KUKA KRL program: nplacestr5LS1.src, nplacestr5LS1.dat

--- nplacestr5LS1.src ---
&ACCESS RVP
&REL 1
&PARAM TEMPLATE = C:\KRC\Roboter\Template\ExpertVorgabe
&PARAM EDITMASK = *
DEF nplacestr5LS1( )
;FOLD INI
  ;FOLD BASISTECH INI
    GLOBAL INTERRUPT DECL 3 WHEN $STOPMESS==TRUE DO IR_STOPM ( )
    INTERRUPT ON 3
    BAS (#INITMOV,0 )
  ;ENDFOLD (BASISTECH INI)
  ;FOLD USER INI
    ;Make your modifications here

  ;ENDFOLD (USER INI)
;ENDFOLD (INI)




SWITCH NumCuring

;*******************************************************
CASE 90501
;*******************************************************
;*** Utilizar para hacer touchup en ptp a continuacion ***;
; 1  Ejecutar Axis_Rob_Move
; 2  Hacer TouchUp en ptp
; 3  Eliminar Axis_Rob_Move y comentarios

Axis_Rob_Move(1.69,-82.8,66.93,14.32,12.14,193,70,50)

;FOLD PTP pWB90501LS1 Vel=100 % PDAT_MESA Tool[10]:AMF1_G1000 Base[14]:BWB2S1;%{PE}%R 5.5.32,%MKUKATPBASIS,%CMOVE,%VPTP,%P 1:PTP, 2:pWB90501LS1, 3:, 5:100, 7:PDAT_MESA
$BWDSTART=FALSE
PDAT_ACT=PPDAT_MESA
FDAT_ACT=FpWB90501LS1
BAS(#PTP_PARAMS,100)
PTP XpWB90501LS1
;ENDFOLD
;*********************************************************;

;***Axis_Rob_Move de ayuda para aproximarse a dejada ***;
; Borrar tras touchup en LIN de dejada
Axis_Rob_Move(-90.22,-57.13,49.23,-5.44,97.37,193.9,20,50)
;*******************************************************;

PTP_OFFS(XP90501LS1, FP90501LS1, 0, -450, 30, 0, 0, 0, #TOOL, 20, 50, 0.0)

Cicle_Grp_M1000 (Inic_Pla_Right)

;***borrar***;
cyltopos(prg_200)
halt
;************;

LIN_OFFS(XP90501LS1, FP90501LS1, 0, 0, 30, 0, 0, 0, #TOOL, 0.1, 50, 0.0)
LIN_OFFS(XP90501LS1, FP90501LS1, 0, 0, 15, 0, 0, 0, #TOOL, 0.1, 50, 0.0)

Cntr_Grp_M1000 (C05C06,RH)

;FOLD LIN P90501LS1 Vel=0.1 m/s LV020Z0 Tool[10]:AMF1_G1000 Base[14]:BWB2S1;%{PE}%R 5.5.32,%MKUKATPBASIS,%CMOVE,%VLIN,%P 1:LIN, 2:P90501LS1, 3:, 5:0.1, 7:V020Z0
$BWDSTART=FALSE
LDAT_ACT=LV020Z0
FDAT_ACT=FP90501LS1
BAS(#CP_PARAMS,0.1)
LIN XP90501LS1
;ENDFOLD

Cntr_Grp_M1000 (AMF09,RLS)
Cyltopos (PRG_51)
Cntr_Grp_M1000 (C07C08,RH)
Cyltopos (PRG_61)
Cntr_Grp_M1000 (AMF10,RLS)
Cntr_Grp_M1000 (C05C06,FREE)
Cntr_Grp_M1000 (C07C08,FREE)
Cyltopos(PRG_88)
LIN_REL{Z -20}#TOOL
Cyltopos (PRG_105)
LIN_REL{Z -30}#TOOL
Cyltopos (PRG_200)

;*** MOVIMIENTOS DE OFFSETS ***;

LIN_OFFS(XP90501LS1, FP90501LS1, 0, 0, -50, 0, 0, 0, #TOOL, 0.3, 50, 0.0)
LIN_OFFS(XP90501LS1, FP90501LS1, 0, -450, -50, 0, 0, 0, #TOOL, 0.3, 50, 0.0)


;******* MEDICION LASER *******;

LIN_OFFS(XPLAS90501LS1_1, FPLAS90501LS1_1, 0, -200, 0, 0, 0, 0, #TOOL, 0.3, 50, 0.0)

cyltopos (prg_61)

;FOLD LIN PLAS90501LS1_1 Vel=0.3 m/s LV020Z0 Tool[10]:AMF1_G1000 Base[14]:BWB2S1;%{PE}%R 5.5.32,%MKUKATPBASIS,%CMOVE,%VLIN,%P 1:LIN, 2:PLAS90501LS1_1, 3:, 5:0.3, 7:V020Z0
$BWDSTART=FALSE
LDAT_ACT=LV020Z0
FDAT_ACT=FPLAS90501LS1_1
BAS(#CP_PARAMS,0.3)
LIN XPLAS90501LS1_1
;ENDFOLD

;Movimimiento de busqueda con laser
;Search( , )

;FOLD LIN PLAS90501LS1_2 Vel=0.3 m/s LV020Z0 Tool[10]:AMF1_G1000 Base[14]:BWB2S1;%{PE}%R 5.5.32,%MKUKATPBASIS,%CMOVE,%VLIN,%P 1:LIN, 2:PLAS90501LS1_2, 3:, 5:0.3, 7:V020Z0
$BWDSTART=FALSE
LDAT_ACT=LV020Z0
FDAT_ACT=FPLAS90501LS1_2
BAS(#CP_PARAMS,0.3)
LIN XPLAS90501LS1_2
;ENDFOLD


;Movimimiento de busqueda con laser
;Search( , )

LIN_OFFS(XPLAS90501LS1_1, FPLAS90501LS1_1, 0, -200, 0, 0, 0, 0, #TOOL, 0.3, 50, 0.0)

;******************************;

;FOLD PTP pWB90501LS1 Vel=100 % PDAT_MESA Tool[10]:AMF1_G1000 Base[14]:BWB2S1;%{PE}%R 5.5.32,%MKUKATPBASIS,%CMOVE,%VPTP,%P 1:PTP, 2:pWB90501LS1, 3:, 5:100, 7:PDAT_MESA
$BWDSTART=FALSE
PDAT_ACT=PPDAT_MESA
FDAT_ACT=FpWB90501LS1
BAS(#PTP_PARAMS,100)
PTP XpWB90501LS1
;ENDFOLD

;*******************************************************
CASE 90503
;*******************************************************
;*** Utilizar para hacer touchup en ptp a continuacion ***;
; 1  Ejecutar Axis_Rob_Move
; 2  Hacer TouchUp en ptp
; 3  Eliminar Axis_Rob_Move y comentarios

Axis_Rob_Move(1.69,-82.8,66.93,14.32,12.14,193,70,50)

;FOLD PTP pWB90503LS1 Vel=100 % PDAT_MESA Tool[10]:AMF1_G1000 Base[14]:BWB2S1;%{PE}%R 5.5.32,%MKUKATPBASIS,%CMOVE,%VPTP,%P 1:PTP, 2:pWB90503LS1, 3:, 5:100, 7:PDAT_MESA
$BWDSTART=FALSE
PDAT_ACT=PPDAT_MESA
FDAT_ACT=FpWB90503LS1
BAS(#PTP_PARAMS,100)
PTP XpWB90503LS1
;ENDFOLD
;*********************************************************;

;***Axis_Rob_Move de ayuda para aproximarse a dejada ***;
; Borrar tras touchup en LIN de dejada
Axis_Rob_Move(-90.22,-57.13,49.23,-5.44,97.37,193.9,20,50)
;*******************************************************;

PTP_OFFS(XP90503LS1, FP90503LS1, 0, -450, 30, 0, 0, 0, #TOOL, 20, 50, 0.0)

Cicle_Grp_M1000 (Inic_Pla_Right)

;***borrar***;
cyltopos(prg_200)
halt
;************;

LIN_OFFS(XP90503LS1, FP90503LS1, 0, 0, 30, 0, 0, 0, #TOOL, 0.1, 50, 0.0)
LIN_OFFS(XP90503LS1, FP90503LS1, 0, 0, 15, 0, 0, 0, #TOOL, 0.1, 50, 0.0)

Cntr_Grp_M1000 (C05C06,RH)

;FOLD LIN P90503LS1 Vel=0.1 m/s LV020Z0 Tool[10]:AMF1_G1000 Base[14]:BWB2S1;%{PE}%R 5.5.32,%MKUKATPBASIS,%CMOVE,%VLIN,%P 1:LIN, 2:P90503LS1, 3:, 5:0.1, 7:V020Z0
$BWDSTART=FALSE
LDAT_ACT=LV020Z0
FDAT_ACT=FP90503LS1
BAS(#CP_PARAMS,0.1)
LIN XP90503LS1
;ENDFOLD

Cntr_Grp_M1000 (AMF09,RLS)
Cyltopos (PRG_51)
Cntr_Grp_M1000 (C07C08,RH)
Cyltopos (PRG_61)
Cntr_Grp_M1000 (AMF10,RLS)
Cntr_Grp_M1000 (C05C06,FREE)
Cntr_Grp_M1000 (C07C08,FREE)
Cyltopos(PRG_88)
LIN_REL{Z -20}#TOOL
Cyltopos (PRG_105)
LIN_REL{Z -30}#TOOL
Cyltopos (PRG_200)

;*** MOVIMIENTOS DE OFFSETS ***;

LIN_OFFS(XP90503LS1, FP90503LS1, 0, 0, -50, 0, 0, 0, #TOOL, 0.3, 50, 0.0)
LIN_OFFS(XP90503LS1, FP90503LS1, 0, -450, -50, 0, 0, 0, #TOOL, 0.3, 50, 0.0)


;******* MEDICION LASER *******;

LIN_OFFS(XPLAS90503LS1_1, FPLAS90503LS1_1, 0, -200, 0, 0, 0, 0, #TOOL, 0.3, 50, 0.0)

cyltopos (prg_61)

;FOLD LIN PLAS90503LS1_1 Vel=0.3 m/s LV020Z0 Tool[10]:AMF1_G1000 Base[14]:BWB2S1;%{PE}%R 5.5.32,%MKUKATPBASIS,%CMOVE,%VLIN,%P 1:LIN, 2:PLAS90503LS1_1, 3:, 5:0.3, 7:V020Z0
$BWDSTART=FALSE
LDAT_ACT=LV020Z0
FDAT_ACT=FPLAS90503LS1_1
BAS(#CP_PARAMS,0.3)
LIN XPLAS90503LS1_1
;ENDFOLD

;Movimimiento de busqueda con laser
;Search( , )

;FOLD LIN PLAS90503LS1_2 Vel=0.3 m/s LV020Z0 Tool[10]:AMF1_G1000 Base[14]:BWB2S1;%{PE}%R 5.5.32,%MKUKATPBASIS,%CMOVE,%VLIN,%P 1:LIN, 2:PLAS90503LS1_2, 3:, 5:0.3, 7:V020Z0
$BWDSTART=FALSE
LDAT_ACT=LV020Z0
FDAT_ACT=FPLAS90503LS1_2
BAS(#CP_PARAMS,0.3)
LIN XPLAS90503LS1_2
;ENDFOLD


;Movimimiento de busqueda con laser
;Search( , )

LIN_OFFS(XPLAS90503LS1_1, FPLAS90503LS1_1, 0, -200, 0, 0, 0, 0, #TOOL, 0.3, 50, 0.0)

;******************************;

;FOLD PTP pWB90503LS1 Vel=100 % PDAT_MESA Tool[10]:AMF1_G1000 Base[14]:BWB2S1;%{PE}%R 5.5.32,%MKUKATPBASIS,%CMOVE,%VPTP,%P 1:PTP, 2:pWB90503LS1, 3:, 5:100, 7:PDAT_MESA
$BWDSTART=FALSE
PDAT_ACT=PPDAT_MESA
FDAT_ACT=FpWB90503LS1
BAS(#PTP_PARAMS,100)
PTP XpWB90503LS1
;ENDFOLD

;*******************************************************
CASE 90505
;*******************************************************
;*** Utilizar para hacer touchup en ptp a continuacion ***;
; 1  Ejecutar Axis_Rob_Move
; 2  Hacer TouchUp en ptp
; 3  Eliminar Axis_Rob_Move y comentarios

Axis_Rob_Move(1.69,-82.8,66.93,14.32,12.14,193,70,50)

;FOLD PTP pWB90505LS1 Vel=100 % PDAT_MESA Tool[10]:AMF1_G1000 Base[14]:BWB2S1;%{PE}%R 5.5.32,%MKUKATPBASIS,%CMOVE,%VPTP,%P 1:PTP, 2:pWB90505LS1, 3:, 5:100, 7:PDAT_MESA
$BWDSTART=FALSE
PDAT_ACT=PPDAT_MESA
FDAT_ACT=FpWB90505LS1
BAS(#PTP_PARAMS,100)
PTP XpWB90505LS1
;ENDFOLD
;*********************************************************;

;***Axis_Rob_Move de ayuda para aproximarse a dejada ***;
; Borrar tras touchup en LIN de dejada
Axis_Rob_Move(-90.22,-57.13,49.23,-5.44,97.37,193.9,20,50)
;*******************************************************;

PTP_OFFS(XP90505LS1, FP90505LS1, 0, -450, 30, 0, 0, 0, #TOOL, 20, 50, 0.0)

Cicle_Grp_M1000 (Inic_Pla_Right)

;***borrar***;
cyltopos(prg_200)
halt
;************;

LIN_OFFS(XP90505LS1, FP90505LS1, 0, 0, 30, 0, 0, 0, #TOOL, 0.1, 50, 0.0)
LIN_OFFS(XP90505LS1, FP90505LS1, 0, 0, 15, 0, 0, 0, #TOOL, 0.1, 50, 0.0)

Cntr_Grp_M1000 (C05C06,RH)

;FOLD LIN P90505LS1 Vel=0.1 m/s LV020Z0 Tool[10]:AMF1_G1000 Base[14]:BWB2S1;%{PE}%R 5.5.32,%MKUKATPBASIS,%CMOVE,%VLIN,%P 1:LIN, 2:P90505LS1, 3:, 5:0.1, 7:V020Z0
$BWDSTART=FALSE
LDAT_ACT=LV020Z0
FDAT_ACT=FP90505LS1
BAS(#CP_PARAMS,0.1)
LIN XP90505LS1
;ENDFOLD

Cntr_Grp_M1000 (AMF09,RLS)
Cyltopos (PRG_51)
Cntr_Grp_M1000 (C07C08,RH)
Cyltopos (PRG_61)
Cntr_Grp_M1000 (AMF10,RLS)
Cntr_Grp_M1000 (C05C06,FREE)
Cntr_Grp_M1000 (C07C08,FREE)
Cyltopos(PRG_88)
LIN_REL{Z -20}#TOOL
Cyltopos (PRG_105)
LIN_REL{Z -30}#TOOL
Cyltopos (PRG_200)

;*** MOVIMIENTOS DE OFFSETS ***;

LIN_OFFS(XP90505LS1, FP90505LS1, 0, 0, -50, 0, 0, 0, #TOOL, 0.3, 50, 0.0)
LIN_OFFS(XP90505LS1, FP90505LS1, 0, -450, -50, 0, 0, 0, #TOOL, 0.3, 50, 0.0)


;******* MEDICION LASER *******;

LIN_OFFS(XPLAS90505LS1_1, FPLAS90505LS1_1, 0, -200, 0, 0, 0, 0, #TOOL, 0.3, 50, 0.0)

cyltopos (prg_61)

;FOLD LIN PLAS90505LS1_1 Vel=0.3 m/s LV020Z0 Tool[10]:AMF1_G1000 Base[14]:BWB2S1;%{PE}%R 5.5.32,%MKUKATPBASIS,%CMOVE,%VLIN,%P 1:LIN, 2:PLAS90505LS1_1, 3:, 5:0.3, 7:V020Z0
$BWDSTART=FALSE
LDAT_ACT=LV020Z0
FDAT_ACT=FPLAS90505LS1_1
BAS(#CP_PARAMS,0.3)
LIN XPLAS90505LS1_1
;ENDFOLD

;Movimimiento de busqueda con laser
;Search( , )

;FOLD LIN PLAS90505LS1_2 Vel=0.3 m/s LV020Z0 Tool[10]:AMF1_G1000 Base[14]:BWB2S1;%{PE}%R 5.5.32,%MKUKATPBASIS,%CMOVE,%VLIN,%P 1:LIN, 2:PLAS90505LS1_2, 3:, 5:0.3, 7:V020Z0
$BWDSTART=FALSE
LDAT_ACT=LV020Z0
FDAT_ACT=FPLAS90505LS1_2
BAS(#CP_PARAMS,0.3)
LIN XPLAS90505LS1_2
;ENDFOLD


;Movimimiento de busqueda con laser
;Search( , )

LIN_OFFS(XPLAS90505LS1_1, FPLAS90505LS1_1, 0, -200, 0, 0, 0, 0, #TOOL, 0.3, 50, 0.0)

;******************************;

;FOLD PTP pWB90505LS1 Vel=100 % PDAT_MESA Tool[10]:AMF1_G1000 Base[14]:BWB2S1;%{PE}%R 5.5.32,%MKUKATPBASIS,%CMOVE,%VPTP,%P 1:PTP, 2:pWB90505LS1, 3:, 5:100, 7:PDAT_MESA
$BWDSTART=FALSE
PDAT_ACT=PPDAT_MESA
FDAT_ACT=FpWB90505LS1
BAS(#PTP_PARAMS,100)
PTP XpWB90505LS1
;ENDFOLD

;*******************************************************
CASE 90507
;*******************************************************
;*** Utilizar para hacer touchup en ptp a continuacion ***;
; 1  Ejecutar Axis_Rob_Move
; 2  Hacer TouchUp en ptp
; 3  Eliminar Axis_Rob_Move y comentarios

Axis_Rob_Move(1.69,-82.8,66.93,14.32,12.14,193,70,50)

;FOLD PTP pWB90507LS1 Vel=100 % PDAT_MESA Tool[10]:AMF1_G1000 Base[14]:BWB2S1;%{PE}%R 5.5.32,%MKUKATPBASIS,%CMOVE,%VPTP,%P 1:PTP, 2:pWB90507LS1, 3:, 5:100, 7:PDAT_MESA
$BWDSTART=FALSE
PDAT_ACT=PPDAT_MESA
FDAT_ACT=FpWB90507LS1
BAS(#PTP_PARAMS,100)
PTP XpWB90507LS1
;ENDFOLD
;*********************************************************;

;***Axis_Rob_Move de ayuda para aproximarse a dejada ***;
; Borrar tras touchup en LIN de dejada
Axis_Rob_Move(-90.22,-57.13,49.23,-5.44,97.37,193.9,20,50)
;*******************************************************;

PTP_OFFS(XP90507LS1, FP90507LS1, 0, -450, 30, 0, 0, 0, #TOOL, 20, 50, 0.0)

Cicle_Grp_M1000 (Inic_Pla_Right)

;***borrar***;
cyltopos(prg_200)
halt
;************;

LIN_OFFS(XP90507LS1, FP90507LS1, 0, 0, 30, 0, 0, 0, #TOOL, 0.1, 50, 0.0)
LIN_OFFS(XP90507LS1, FP90507LS1, 0, 0, 15, 0, 0, 0, #TOOL, 0.1, 50, 0.0)

Cntr_Grp_M1000 (C05C06,RH)

;FOLD LIN P90507LS1 Vel=0.1 m/s LV020Z0 Tool[10]:AMF1_G1000 Base[14]:BWB2S1;%{PE}%R 5.5.32,%MKUKATPBASIS,%CMOVE,%VLIN,%P 1:LIN, 2:P90507LS1, 3:, 5:0.1, 7:V020Z0
$BWDSTART=FALSE
LDAT_ACT=LV020Z0
FDAT_ACT=FP90507LS1
BAS(#CP_PARAMS,0.1)
LIN XP90507LS1
;ENDFOLD

Cntr_Grp_M1000 (AMF09,RLS)
Cyltopos (PRG_51)
Cntr_Grp_M1000 (C07C08,RH)
Cyltopos (PRG_61)
Cntr_Grp_M1000 (AMF10,RLS)
Cntr_Grp_M1000 (C05C06,FREE)
Cntr_Grp_M1000 (C07C08,FREE)
Cyltopos(PRG_88)
LIN_REL{Z -20}#TOOL
Cyltopos (PRG_105)
LIN_REL{Z -30}#TOOL
Cyltopos (PRG_200)

;*** MOVIMIENTOS DE OFFSETS ***;

LIN_OFFS(XP90507LS1, FP90507LS1, 0, 0, -50, 0, 0, 0, #TOOL, 0.3, 50, 0.0)
LIN_OFFS(XP90507LS1, FP90507LS1, 0, -450, -50, 0, 0, 0, #TOOL, 0.3, 50, 0.0)


;******* MEDICION LASER *******;

LIN_OFFS(XPLAS90507LS1_1, FPLAS90507LS1_1, 0, -200, 0, 0, 0, 0, #TOOL, 0.3, 50, 0.0)

cyltopos (prg_61)

;FOLD LIN PLAS90507LS1_1 Vel=0.3 m/s LV020Z0 Tool[10]:AMF1_G1000 Base[14]:BWB2S1;%{PE}%R 5.5.32,%MKUKATPBASIS,%CMOVE,%VLIN,%P 1:LIN, 2:PLAS90507LS1_1, 3:, 5:0.3, 7:V020Z0
$BWDSTART=FALSE
LDAT_ACT=LV020Z0
FDAT_ACT=FPLAS90507LS1_1
BAS(#CP_PARAMS,0.3)
LIN XPLAS90507LS1_1
;ENDFOLD

;Movimimiento de busqueda con laser
;Search( , )

;FOLD LIN PLAS90507LS1_2 Vel=0.3 m/s LV020Z0 Tool[10]:AMF1_G1000 Base[14]:BWB2S1;%{PE}%R 5.5.32,%MKUKATPBASIS,%CMOVE,%VLIN,%P 1:LIN, 2:PLAS90507LS1_2, 3:, 5:0.3, 7:V020Z0
$BWDSTART=FALSE
LDAT_ACT=LV020Z0
FDAT_ACT=FPLAS90507LS1_2
BAS(#CP_PARAMS,0.3)
LIN XPLAS90507LS1_2
;ENDFOLD


;Movimimiento de busqueda con laser
;Search( , )

LIN_OFFS(XPLAS90507LS1_1, FPLAS90507LS1_1, 0, -200, 0, 0, 0, 0, #TOOL, 0.3, 50, 0.0)

;******************************;

;FOLD PTP pWB90507LS1 Vel=100 % PDAT_MESA Tool[10]:AMF1_G1000 Base[14]:BWB2S1;%{PE}%R 5.5.32,%MKUKATPBASIS,%CMOVE,%VPTP,%P 1:PTP, 2:pWB90507LS1, 3:, 5:100, 7:PDAT_MESA
$BWDSTART=FALSE
PDAT_ACT=PPDAT_MESA
FDAT_ACT=FpWB90507LS1
BAS(#PTP_PARAMS,100)
PTP XpWB90507LS1
;ENDFOLD

;*******************************************************
CASE 90509
;*******************************************************
;*** Utilizar para hacer touchup en ptp a continuacion ***;
; 1  Ejecutar Axis_Rob_Move
; 2  Hacer TouchUp en ptp
; 3  Eliminar Axis_Rob_Move y comentarios

Axis_Rob_Move(1.69,-82.8,66.93,14.32,12.14,193,70,50)

;FOLD PTP pWB90509LS1 Vel=100 % PDAT_MESA Tool[10]:AMF1_G1000 Base[14]:BWB2S1;%{PE}%R 5.5.32,%MKUKATPBASIS,%CMOVE,%VPTP,%P 1:PTP, 2:pWB90509LS1, 3:, 5:100, 7:PDAT_MESA
$BWDSTART=FALSE
PDAT_ACT=PPDAT_MESA
FDAT_ACT=FpWB90509LS1
BAS(#PTP_PARAMS,100)
PTP XpWB90509LS1
;ENDFOLD
;*********************************************************;

;***Axis_Rob_Move de ayuda para aproximarse a dejada ***;
; Borrar tras touchup en LIN de dejada
Axis_Rob_Move(-90.22,-57.13,49.23,-5.44,97.37,193.9,20,50)
;*******************************************************;

PTP_OFFS(XP90509LS1, FP90509LS1, 0, -450, 30, 0, 0, 0, #TOOL, 20, 50, 0.0)

Cicle_Grp_M1000 (Inic_Pla_Right)

;***borrar***;
cyltopos(prg_200)
halt
;************;

LIN_OFFS(XP90509LS1, FP90509LS1, 0, 0, 30, 0, 0, 0, #TOOL, 0.1, 50, 0.0)
LIN_OFFS(XP90509LS1, FP90509LS1, 0, 0, 15, 0, 0, 0, #TOOL, 0.1, 50, 0.0)

Cntr_Grp_M1000 (C05C06,RH)

;FOLD LIN P90509LS1 Vel=0.1 m/s LV020Z0 Tool[10]:AMF1_G1000 Base[14]:BWB2S1;%{PE}%R 5.5.32,%MKUKATPBASIS,%CMOVE,%VLIN,%P 1:LIN, 2:P90509LS1, 3:, 5:0.1, 7:V020Z0
$BWDSTART=FALSE
LDAT_ACT=LV020Z0
FDAT_ACT=FP90509LS1
BAS(#CP_PARAMS,0.1)
LIN XP90509LS1
;ENDFOLD

Cntr_Grp_M1000 (AMF09,RLS)
Cyltopos (PRG_51)
Cntr_Grp_M1000 (C07C08,RH)
Cyltopos (PRG_61)
Cntr_Grp_M1000 (AMF10,RLS)
Cntr_Grp_M1000 (C05C06,FREE)
Cntr_Grp_M1000 (C07C08,FREE)
Cyltopos(PRG_88)
LIN_REL{Z -20}#TOOL
Cyltopos (PRG_105)
LIN_REL{Z -30}#TOOL
Cyltopos (PRG_200)

;*** MOVIMIENTOS DE OFFSETS ***;

LIN_OFFS(XP90509LS1, FP90509LS1, 0, 0, -50, 0, 0, 0, #TOOL, 0.3, 50, 0.0)
LIN_OFFS(XP90509LS1, FP90509LS1, 0, -450, -50, 0, 0, 0, #TOOL, 0.3, 50, 0.0)


;******* MEDICION LASER *******;

LIN_OFFS(XPLAS90509LS1_1, FPLAS90509LS1_1, 0, -200, 0, 0, 0, 0, #TOOL, 0.3, 50, 0.0)

cyltopos (prg_61)

;FOLD LIN PLAS90509LS1_1 Vel=0.3 m/s LV020Z0 Tool[10]:AMF1_G1000 Base[14]:BWB2S1;%{PE}%R 5.5.32,%MKUKATPBASIS,%CMOVE,%VLIN,%P 1:LIN, 2:PLAS90509LS1_1, 3:, 5:0.3, 7:V020Z0
$BWDSTART=FALSE
LDAT_ACT=LV020Z0
FDAT_ACT=FPLAS90509LS1_1
BAS(#CP_PARAMS,0.3)
LIN XPLAS90509LS1_1
;ENDFOLD

;Movimimiento de busqueda con laser
;Search( , )

;FOLD LIN PLAS90509LS1_2 Vel=0.3 m/s LV020Z0 Tool[10]:AMF1_G1000 Base[14]:BWB2S1;%{PE}%R 5.5.32,%MKUKATPBASIS,%CMOVE,%VLIN,%P 1:LIN, 2:PLAS90509LS1_2, 3:, 5:0.3, 7:V020Z0
$BWDSTART=FALSE
LDAT_ACT=LV020Z0
FDAT_ACT=FPLAS90509LS1_2
BAS(#CP_PARAMS,0.3)
LIN XPLAS90509LS1_2
;ENDFOLD


;Movimimiento de busqueda con laser
;Search( , )

LIN_OFFS(XPLAS90509LS1_1, FPLAS90509LS1_1, 0, -200, 0, 0, 0, 0, #TOOL, 0.3, 50, 0.0)

;******************************;

;FOLD PTP pWB90509LS1 Vel=100 % PDAT_MESA Tool[10]:AMF1_G1000 Base[14]:BWB2S1;%{PE}%R 5.5.32,%MKUKATPBASIS,%CMOVE,%VPTP,%P 1:PTP, 2:pWB90509LS1, 3:, 5:100, 7:PDAT_MESA
$BWDSTART=FALSE
PDAT_ACT=PPDAT_MESA
FDAT_ACT=FpWB90509LS1
BAS(#PTP_PARAMS,100)
PTP XpWB90509LS1
;ENDFOLD

;*******************************************************
CASE 90511
;*******************************************************
;*** Utilizar para hacer touchup en ptp a continuacion ***;
; 1  Ejecutar Axis_Rob_Move
; 2  Hacer TouchUp en ptp
; 3  Eliminar Axis_Rob_Move y comentarios

Axis_Rob_Move(1.69,-82.8,66.93,14.32,12.14,193,70,50)

;FOLD PTP pWB90511LS1 Vel=100 % PDAT_MESA Tool[10]:AMF1_G1000 Base[14]:BWB2S1;%{PE}%R 5.5.32,%MKUKATPBASIS,%CMOVE,%VPTP,%P 1:PTP, 2:pWB90511LS1, 3:, 5:100, 7:PDAT_MESA
$BWDSTART=FALSE
PDAT_ACT=PPDAT_MESA
FDAT_ACT=FpWB90511LS1
BAS(#PTP_PARAMS,100)
PTP XpWB90511LS1
;ENDFOLD
;*********************************************************;

;***Axis_Rob_Move de ayuda para aproximarse a dejada ***;
; Borrar tras touchup en LIN de dejada
Axis_Rob_Move(-90.22,-57.13,49.23,-5.44,97.37,193.9,20,50)
;*******************************************************;

PTP_OFFS(XP90511LS1, FP90511LS1, 0, -450, 30, 0, 0, 0, #TOOL, 20, 50, 0.0)

Cicle_Grp_M1000 (Inic_Pla_Right)

;***borrar***;
cyltopos(prg_200)
halt
;************;

LIN_OFFS(XP90511LS1, FP90511LS1, 0, 0, 30, 0, 0, 0, #TOOL, 0.1, 50, 0.0)
LIN_OFFS(XP90511LS1, FP90511LS1, 0, 0, 15, 0, 0, 0, #TOOL, 0.1, 50, 0.0)

Cntr_Grp_M1000 (C05C06,RH)

;FOLD LIN P90511LS1 Vel=0.1 m/s LV020Z0 Tool[10]:AMF1_G1000 Base[14]:BWB2S1;%{PE}%R 5.5.32,%MKUKATPBASIS,%CMOVE,%VLIN,%P 1:LIN, 2:P90511LS1, 3:, 5:0.1, 7:V020Z0
$BWDSTART=FALSE
LDAT_ACT=LV020Z0
FDAT_ACT=FP90511LS1
BAS(#CP_PARAMS,0.1)
LIN XP90511LS1
;ENDFOLD

Cntr_Grp_M1000 (AMF09,RLS)
Cyltopos (PRG_51)
Cntr_Grp_M1000 (C07C08,RH)
Cyltopos (PRG_61)
Cntr_Grp_M1000 (AMF10,RLS)
Cntr_Grp_M1000 (C05C06,FREE)
Cntr_Grp_M1000 (C07C08,FREE)
Cyltopos(PRG_88)
LIN_REL{Z -20}#TOOL
Cyltopos (PRG_105)
LIN_REL{Z -30}#TOOL
Cyltopos (PRG_200)

;*** MOVIMIENTOS DE OFFSETS ***;

LIN_OFFS(XP90511LS1, FP90511LS1, 0, 0, -50, 0, 0, 0, #TOOL, 0.3, 50, 0.0)
LIN_OFFS(XP90511LS1, FP90511LS1, 0, -450, -50, 0, 0, 0, #TOOL, 0.3, 50, 0.0)


;******* MEDICION LASER *******;

LIN_OFFS(XPLAS90511LS1_1, FPLAS90511LS1_1, 0, -200, 0, 0, 0, 0, #TOOL, 0.3, 50, 0.0)

cyltopos (prg_61)

;FOLD LIN PLAS90511LS1_1 Vel=0.3 m/s LV020Z0 Tool[10]:AMF1_G1000 Base[14]:BWB2S1;%{PE}%R 5.5.32,%MKUKATPBASIS,%CMOVE,%VLIN,%P 1:LIN, 2:PLAS90511LS1_1, 3:, 5:0.3, 7:V020Z0
$BWDSTART=FALSE
LDAT_ACT=LV020Z0
FDAT_ACT=FPLAS90511LS1_1
BAS(#CP_PARAMS,0.3)
LIN XPLAS90511LS1_1
;ENDFOLD

;Movimimiento de busqueda con laser
;Search( , )

;FOLD LIN PLAS90511LS1_2 Vel=0.3 m/s LV020Z0 Tool[10]:AMF1_G1000 Base[14]:BWB2S1;%{PE}%R 5.5.32,%MKUKATPBASIS,%CMOVE,%VLIN,%P 1:LIN, 2:PLAS90511LS1_2, 3:, 5:0.3, 7:V020Z0
$BWDSTART=FALSE
LDAT_ACT=LV020Z0
FDAT_ACT=FPLAS90511LS1_2
BAS(#CP_PARAMS,0.3)
LIN XPLAS90511LS1_2
;ENDFOLD


;Movimimiento de busqueda con laser
;Search( , )

LIN_OFFS(XPLAS90511LS1_1, FPLAS90511LS1_1, 0, -200, 0, 0, 0, 0, #TOOL, 0.3, 50, 0.0)

;******************************;

;FOLD PTP pWB90511LS1 Vel=100 % PDAT_MESA Tool[10]:AMF1_G1000 Base[14]:BWB2S1;%{PE}%R 5.5.32,%MKUKATPBASIS,%CMOVE,%VPTP,%P 1:PTP, 2:pWB90511LS1, 3:, 5:100, 7:PDAT_MESA
$BWDSTART=FALSE
PDAT_ACT=PPDAT_MESA
FDAT_ACT=FpWB90511LS1
BAS(#PTP_PARAMS,100)
PTP XpWB90511LS1
;ENDFOLD

;*******************************************************
CASE 90513
;*******************************************************
;*** Utilizar para hacer touchup en ptp a continuacion ***;
; 1  Ejecutar Axis_Rob_Move
; 2  Hacer TouchUp en ptp
; 3  Eliminar Axis_Rob_Move y comentarios

Axis_Rob_Move(1.69,-82.8,66.93,14.32,12.14,193,70,50)

;FOLD PTP pWB90513LS1 Vel=100 % PDAT_MESA Tool[10]:AMF1_G1000 Base[14]:BWB2S1;%{PE}%R 5.5.32,%MKUKATPBASIS,%CMOVE,%VPTP,%P 1:PTP, 2:pWB90513LS1, 3:, 5:100, 7:PDAT_MESA
$BWDSTART=FALSE
PDAT_ACT=PPDAT_MESA
FDAT_ACT=FpWB90513LS1
BAS(#PTP_PARAMS,100)
PTP XpWB90513LS1
;ENDFOLD
;*********************************************************;

;***Axis_Rob_Move de ayuda para aproximarse a dejada ***;
; Borrar tras touchup en LIN de dejada
Axis_Rob_Move(-90.22,-57.13,49.23,-5.44,97.37,193.9,20,50)
;*******************************************************;

PTP_OFFS(XP90513LS1, FP90513LS1, 0, -450, 30, 0, 0, 0, #TOOL, 20, 50, 0.0)

Cicle_Grp_M1000 (Inic_Pla_Right)

;***borrar***;
cyltopos(prg_200)
halt
;************;

LIN_OFFS(XP90513LS1, FP90513LS1, 0, 0, 30, 0, 0, 0, #TOOL, 0.1, 50, 0.0)
LIN_OFFS(XP90513LS1, FP90513LS1, 0, 0, 15, 0, 0, 0, #TOOL, 0.1, 50, 0.0)

Cntr_Grp_M1000 (C05C06,RH)

;FOLD LIN P90513LS1 Vel=0.1 m/s LV020Z0 Tool[10]:AMF1_G1000 Base[14]:BWB2S1;%{PE}%R 5.5.32,%MKUKATPBASIS,%CMOVE,%VLIN,%P 1:LIN, 2:P90513LS1, 3:, 5:0.1, 7:V020Z0
$BWDSTART=FALSE
LDAT_ACT=LV020Z0
FDAT_ACT=FP90513LS1
BAS(#CP_PARAMS,0.1)
LIN XP90513LS1
;ENDFOLD

Cntr_Grp_M1000 (AMF09,RLS)
Cyltopos (PRG_51)
Cntr_Grp_M1000 (C07C08,RH)
Cyltopos (PRG_61)
Cntr_Grp_M1000 (AMF10,RLS)
Cntr_Grp_M1000 (C05C06,FREE)
Cntr_Grp_M1000 (C07C08,FREE)
Cyltopos(PRG_88)
LIN_REL{Z -20}#TOOL
Cyltopos (PRG_105)
LIN_REL{Z -30}#TOOL
Cyltopos (PRG_200)

;*** MOVIMIENTOS DE OFFSETS ***;

LIN_OFFS(XP90513LS1, FP90513LS1, 0, 0, -50, 0, 0, 0, #TOOL, 0.3, 50, 0.0)
LIN_OFFS(XP90513LS1, FP90513LS1, 0, -450, -50, 0, 0, 0, #TOOL, 0.3, 50, 0.0)


;******* MEDICION LASER *******;

LIN_OFFS(XPLAS90513LS1_1, FPLAS90513LS1_1, 0, -200, 0, 0, 0, 0, #TOOL, 0.3, 50, 0.0)

cyltopos (prg_61)

;FOLD LIN PLAS90513LS1_1 Vel=0.3 m/s LV020Z0 Tool[10]:AMF1_G1000 Base[14]:BWB2S1;%{PE}%R 5.5.32,%MKUKATPBASIS,%CMOVE,%VLIN,%P 1:LIN, 2:PLAS90513LS1_1, 3:, 5:0.3, 7:V020Z0
$BWDSTART=FALSE
LDAT_ACT=LV020Z0
FDAT_ACT=FPLAS90513LS1_1
BAS(#CP_PARAMS,0.3)
LIN XPLAS90513LS1_1
;ENDFOLD

;Movimimiento de busqueda con laser
;Search( , )

;FOLD LIN PLAS90513LS1_2 Vel=0.3 m/s LV020Z0 Tool[10]:AMF1_G1000 Base[14]:BWB2S1;%{PE}%R 5.5.32,%MKUKATPBASIS,%CMOVE,%VLIN,%P 1:LIN, 2:PLAS90513LS1_2, 3:, 5:0.3, 7:V020Z0
$BWDSTART=FALSE
LDAT_ACT=LV020Z0
FDAT_ACT=FPLAS90513LS1_2
BAS(#CP_PARAMS,0.3)
LIN XPLAS90513LS1_2
;ENDFOLD


;Movimimiento de busqueda con laser
;Search( , )

LIN_OFFS(XPLAS90513LS1_1, FPLAS90513LS1_1, 0, -200, 0, 0, 0, 0, #TOOL, 0.3, 50, 0.0)

;******************************;

;FOLD PTP pWB90513LS1 Vel=100 % PDAT_MESA Tool[10]:AMF1_G1000 Base[14]:BWB2S1;%{PE}%R 5.5.32,%MKUKATPBASIS,%CMOVE,%VPTP,%P 1:PTP, 2:pWB90513LS1, 3:, 5:100, 7:PDAT_MESA
$BWDSTART=FALSE
PDAT_ACT=PPDAT_MESA
FDAT_ACT=FpWB90513LS1
BAS(#PTP_PARAMS,100)
PTP XpWB90513LS1
;ENDFOLD

;*******************************************************
CASE 90515
;*******************************************************
;*** Utilizar para hacer touchup en ptp a continuacion ***;
; 1  Ejecutar Axis_Rob_Move
; 2  Hacer TouchUp en ptp
; 3  Eliminar Axis_Rob_Move y comentarios

Axis_Rob_Move(1.69,-82.8,66.93,14.32,12.14,193,70,50)

;FOLD PTP pWB90515LS1 Vel=100 % PDAT_MESA Tool[10]:AMF1_G1000 Base[14]:BWB2S1;%{PE}%R 5.5.32,%MKUKATPBASIS,%CMOVE,%VPTP,%P 1:PTP, 2:pWB90515LS1, 3:, 5:100, 7:PDAT_MESA
$BWDSTART=FALSE
PDAT_ACT=PPDAT_MESA
FDAT_ACT=FpWB90515LS1
BAS(#PTP_PARAMS,100)
PTP XpWB90515LS1
;ENDFOLD
;*********************************************************;

;***Axis_Rob_Move de ayuda para aproximarse a dejada ***;
; Borrar tras touchup en LIN de dejada
Axis_Rob_Move(-90.22,-57.13,49.23,-5.44,97.37,193.9,20,50)
;*******************************************************;

PTP_OFFS(XP90515LS1, FP90515LS1, 0, -450, 30, 0, 0, 0, #TOOL, 20, 50, 0.0)

Cicle_Grp_M1000 (Inic_Pla_Right)

;***borrar***;
cyltopos(prg_200)
halt
;************;

LIN_OFFS(XP90515LS1, FP90515LS1, 0, 0, 30, 0, 0, 0, #TOOL, 0.1, 50, 0.0)
LIN_OFFS(XP90515LS1, FP90515LS1, 0, 0, 15, 0, 0, 0, #TOOL, 0.1, 50, 0.0)

Cntr_Grp_M1000 (C05C06,RH)

;FOLD LIN P90515LS1 Vel=0.1 m/s LV020Z0 Tool[10]:AMF1_G1000 Base[14]:BWB2S1;%{PE}%R 5.5.32,%MKUKATPBASIS,%CMOVE,%VLIN,%P 1:LIN, 2:P90515LS1, 3:, 5:0.1, 7:V020Z0
$BWDSTART=FALSE
LDAT_ACT=LV020Z0
FDAT_ACT=FP90515LS1
BAS(#CP_PARAMS,0.1)
LIN XP90515LS1
;ENDFOLD

Cntr_Grp_M1000 (AMF09,RLS)
Cyltopos (PRG_51)
Cntr_Grp_M1000 (C07C08,RH)
Cyltopos (PRG_61)
Cntr_Grp_M1000 (AMF10,RLS)
Cntr_Grp_M1000 (C05C06,FREE)
Cntr_Grp_M1000 (C07C08,FREE)
Cyltopos(PRG_88)
LIN_REL{Z -20}#TOOL
Cyltopos (PRG_105)
LIN_REL{Z -30}#TOOL
Cyltopos (PRG_200)

;*** MOVIMIENTOS DE OFFSETS ***;

LIN_OFFS(XP90515LS1, FP90515LS1, 0, 0, -50, 0, 0, 0, #TOOL, 0.3, 50, 0.0)
LIN_OFFS(XP90515LS1, FP90515LS1, 0, -450, -50, 0, 0, 0, #TOOL, 0.3, 50, 0.0)


;******* MEDICION LASER *******;

LIN_OFFS(XPLAS90515LS1_1, FPLAS90515LS1_1, 0, -200, 0, 0, 0, 0, #TOOL, 0.3, 50, 0.0)

cyltopos (prg_61)

;FOLD LIN PLAS90515LS1_1 Vel=0.3 m/s LV020Z0 Tool[10]:AMF1_G1000 Base[14]:BWB2S1;%{PE}%R 5.5.32,%MKUKATPBASIS,%CMOVE,%VLIN,%P 1:LIN, 2:PLAS90515LS1_1, 3:, 5:0.3, 7:V020Z0
$BWDSTART=FALSE
LDAT_ACT=LV020Z0
FDAT_ACT=FPLAS90515LS1_1
BAS(#CP_PARAMS,0.3)
LIN XPLAS90515LS1_1
;ENDFOLD

;Movimimiento de busqueda con laser
;Search( , )

;FOLD LIN PLAS90515LS1_2 Vel=0.3 m/s LV020Z0 Tool[10]:AMF1_G1000 Base[14]:BWB2S1;%{PE}%R 5.5.32,%MKUKATPBASIS,%CMOVE,%VLIN,%P 1:LIN, 2:PLAS90515LS1_2, 3:, 5:0.3, 7:V020Z0
$BWDSTART=FALSE
LDAT_ACT=LV020Z0
FDAT_ACT=FPLAS90515LS1_2
BAS(#CP_PARAMS,0.3)
LIN XPLAS90515LS1_2
;ENDFOLD


;Movimimiento de busqueda con laser
;Search( , )

LIN_OFFS(XPLAS90515LS1_1, FPLAS90515LS1_1, 0, -200, 0, 0, 0, 0, #TOOL, 0.3, 50, 0.0)

;******************************;

;FOLD PTP pWB90515LS1 Vel=100 % PDAT_MESA Tool[10]:AMF1_G1000 Base[14]:BWB2S1;%{PE}%R 5.5.32,%MKUKATPBASIS,%CMOVE,%VPTP,%P 1:PTP, 2:pWB90515LS1, 3:, 5:100, 7:PDAT_MESA
$BWDSTART=FALSE
PDAT_ACT=PPDAT_MESA
FDAT_ACT=FpWB90515LS1
BAS(#PTP_PARAMS,100)
PTP XpWB90515LS1
;ENDFOLD

;*******************************************************
CASE 90517
;*******************************************************
;*** Utilizar para hacer touchup en ptp a continuacion ***;
; 1  Ejecutar Axis_Rob_Move
; 2  Hacer TouchUp en ptp
; 3  Eliminar Axis_Rob_Move y comentarios

Axis_Rob_Move(1.69,-82.8,66.93,14.32,12.14,193,70,50)

;FOLD PTP pWB90517LS1 Vel=100 % PDAT_MESA Tool[10]:AMF1_G1000 Base[14]:BWB2S1;%{PE}%R 5.5.32,%MKUKATPBASIS,%CMOVE,%VPTP,%P 1:PTP, 2:pWB90517LS1, 3:, 5:100, 7:PDAT_MESA
$BWDSTART=FALSE
PDAT_ACT=PPDAT_MESA
FDAT_ACT=FpWB90517LS1
BAS(#PTP_PARAMS,100)
PTP XpWB90517LS1
;ENDFOLD
;*********************************************************;

;***Axis_Rob_Move de ayuda para aproximarse a dejada ***;
; Borrar tras touchup en LIN de dejada
Axis_Rob_Move(-90.22,-57.13,49.23,-5.44,97.37,193.9,20,50)
;*******************************************************;

PTP_OFFS(XP90517LS1, FP90517LS1, 0, -450, 30, 0, 0, 0, #TOOL, 20, 50, 0.0)

Cicle_Grp_M1000 (Inic_Pla_Right)

;***borrar***;
cyltopos(prg_200)
halt
;************;

LIN_OFFS(XP90517LS1, FP90517LS1, 0, 0, 30, 0, 0, 0, #TOOL, 0.1, 50, 0.0)
LIN_OFFS(XP90517LS1, FP90517LS1, 0, 0, 15, 0, 0, 0, #TOOL, 0.1, 50, 0.0)

Cntr_Grp_M1000 (C05C06,RH)

;FOLD LIN P90517LS1 Vel=0.1 m/s LV020Z0 Tool[10]:AMF1_G1000 Base[14]:BWB2S1;%{PE}%R 5.5.32,%MKUKATPBASIS,%CMOVE,%VLIN,%P 1:LIN, 2:P90517LS1, 3:, 5:0.1, 7:V020Z0
$BWDSTART=FALSE
LDAT_ACT=LV020Z0
FDAT_ACT=FP90517LS1
BAS(#CP_PARAMS,0.1)
LIN XP90517LS1
;ENDFOLD

Cntr_Grp_M1000 (AMF09,RLS)
Cyltopos (PRG_51)
Cntr_Grp_M1000 (C07C08,RH)
Cyltopos (PRG_61)
Cntr_Grp_M1000 (AMF10,RLS)
Cntr_Grp_M1000 (C05C06,FREE)
Cntr_Grp_M1000 (C07C08,FREE)
Cyltopos(PRG_88)
LIN_REL{Z -20}#TOOL
Cyltopos (PRG_105)
LIN_REL{Z -30}#TOOL
Cyltopos (PRG_200)

;*** MOVIMIENTOS DE OFFSETS ***;

LIN_OFFS(XP90517LS1, FP90517LS1, 0, 0, -50, 0, 0, 0, #TOOL, 0.3, 50, 0.0)
LIN_OFFS(XP90517LS1, FP90517LS1, 0, -450, -50, 0, 0, 0, #TOOL, 0.3, 50, 0.0)


;******* MEDICION LASER *******;

LIN_OFFS(XPLAS90517LS1_1, FPLAS90517LS1_1, 0, -200, 0, 0, 0, 0, #TOOL, 0.3, 50, 0.0)

cyltopos (prg_61)

;FOLD LIN PLAS90517LS1_1 Vel=0.3 m/s LV020Z0 Tool[10]:AMF1_G1000 Base[14]:BWB2S1;%{PE}%R 5.5.32,%MKUKATPBASIS,%CMOVE,%VLIN,%P 1:LIN, 2:PLAS90517LS1_1, 3:, 5:0.3, 7:V020Z0
$BWDSTART=FALSE
LDAT_ACT=LV020Z0
FDAT_ACT=FPLAS90517LS1_1
BAS(#CP_PARAMS,0.3)
LIN XPLAS90517LS1_1
;ENDFOLD

;Movimimiento de busqueda con laser
;Search( , )

;FOLD LIN PLAS90517LS1_2 Vel=0.3 m/s LV020Z0 Tool[10]:AMF1_G1000 Base[14]:BWB2S1;%{PE}%R 5.5.32,%MKUKATPBASIS,%CMOVE,%VLIN,%P 1:LIN, 2:PLAS90517LS1_2, 3:, 5:0.3, 7:V020Z0
$BWDSTART=FALSE
LDAT_ACT=LV020Z0
FDAT_ACT=FPLAS90517LS1_2
BAS(#CP_PARAMS,0.3)
LIN XPLAS90517LS1_2
;ENDFOLD


;Movimimiento de busqueda con laser
;Search( , )

LIN_OFFS(XPLAS90517LS1_1, FPLAS90517LS1_1, 0, -200, 0, 0, 0, 0, #TOOL, 0.3, 50, 0.0)

;******************************;

;FOLD PTP pWB90517LS1 Vel=100 % PDAT_MESA Tool[10]:AMF1_G1000 Base[14]:BWB2S1;%{PE}%R 5.5.32,%MKUKATPBASIS,%CMOVE,%VPTP,%P 1:PTP, 2:pWB90517LS1, 3:, 5:100, 7:PDAT_MESA
$BWDSTART=FALSE
PDAT_ACT=PPDAT_MESA
FDAT_ACT=FpWB90517LS1
BAS(#PTP_PARAMS,100)
PTP XpWB90517LS1
;ENDFOLD

;*******************************************************
CASE 90519
;*******************************************************
;*** Utilizar para hacer touchup en ptp a continuacion ***;
; 1  Ejecutar Axis_Rob_Move
; 2  Hacer TouchUp en ptp
; 3  Eliminar Axis_Rob_Move y comentarios

Axis_Rob_Move(1.69,-82.8,66.93,14.32,12.14,193,70,50)

;FOLD PTP pWB90519LS1 Vel=100 % PDAT_MESA Tool[10]:AMF1_G1000 Base[14]:BWB2S1;%{PE}%R 5.5.32,%MKUKATPBASIS,%CMOVE,%VPTP,%P 1:PTP, 2:pWB90519LS1, 3:, 5:100, 7:PDAT_MESA
$BWDSTART=FALSE
PDAT_ACT=PPDAT_MESA
FDAT_ACT=FpWB90519LS1
BAS(#PTP_PARAMS,100)
PTP XpWB90519LS1
;ENDFOLD
;*********************************************************;

;***Axis_Rob_Move de ayuda para aproximarse a dejada ***;
; Borrar tras touchup en LIN de dejada
Axis_Rob_Move(-90.22,-57.13,49.23,-5.44,97.37,193.9,20,50)
;*******************************************************;

PTP_OFFS(XP90519LS1, FP90519LS1, 0, -450, 30, 0, 0, 0, #TOOL, 20, 50, 0.0)

Cicle_Grp_M1000 (Inic_Pla_Right)

;***borrar***;
cyltopos(prg_200)
halt
;************;

LIN_OFFS(XP90519LS1, FP90519LS1, 0, 0, 30, 0, 0, 0, #TOOL, 0.1, 50, 0.0)
LIN_OFFS(XP90519LS1, FP90519LS1, 0, 0, 15, 0, 0, 0, #TOOL, 0.1, 50, 0.0)

Cntr_Grp_M1000 (C05C06,RH)

;FOLD LIN P90519LS1 Vel=0.1 m/s LV020Z0 Tool[10]:AMF1_G1000 Base[14]:BWB2S1;%{PE}%R 5.5.32,%MKUKATPBASIS,%CMOVE,%VLIN,%P 1:LIN, 2:P90519LS1, 3:, 5:0.1, 7:V020Z0
$BWDSTART=FALSE
LDAT_ACT=LV020Z0
FDAT_ACT=FP90519LS1
BAS(#CP_PARAMS,0.1)
LIN XP90519LS1
;ENDFOLD

Cntr_Grp_M1000 (AMF09,RLS)
Cyltopos (PRG_51)
Cntr_Grp_M1000 (C07C08,RH)
Cyltopos (PRG_61)
Cntr_Grp_M1000 (AMF10,RLS)
Cntr_Grp_M1000 (C05C06,FREE)
Cntr_Grp_M1000 (C07C08,FREE)
Cyltopos(PRG_88)
LIN_REL{Z -20}#TOOL
Cyltopos (PRG_105)
LIN_REL{Z -30}#TOOL
Cyltopos (PRG_200)

;*** MOVIMIENTOS DE OFFSETS ***;

LIN_OFFS(XP90519LS1, FP90519LS1, 0, 0, -50, 0, 0, 0, #TOOL, 0.3, 50, 0.0)
LIN_OFFS(XP90519LS1, FP90519LS1, 0, -450, -50, 0, 0, 0, #TOOL, 0.3, 50, 0.0)


;******* MEDICION LASER *******;

LIN_OFFS(XPLAS90519LS1_1, FPLAS90519LS1_1, 0, -200, 0, 0, 0, 0, #TOOL, 0.3, 50, 0.0)

cyltopos (prg_61)

;FOLD LIN PLAS90519LS1_1 Vel=0.3 m/s LV020Z0 Tool[10]:AMF1_G1000 Base[14]:BWB2S1;%{PE}%R 5.5.32,%MKUKATPBASIS,%CMOVE,%VLIN,%P 1:LIN, 2:PLAS90519LS1_1, 3:, 5:0.3, 7:V020Z0
$BWDSTART=FALSE
LDAT_ACT=LV020Z0
FDAT_ACT=FPLAS90519LS1_1
BAS(#CP_PARAMS,0.3)
LIN XPLAS90519LS1_1
;ENDFOLD

;Movimimiento de busqueda con laser
;Search( , )

;FOLD LIN PLAS90519LS1_2 Vel=0.3 m/s LV020Z0 Tool[10]:AMF1_G1000 Base[14]:BWB2S1;%{PE}%R 5.5.32,%MKUKATPBASIS,%CMOVE,%VLIN,%P 1:LIN, 2:PLAS90519LS1_2, 3:, 5:0.3, 7:V020Z0
$BWDSTART=FALSE
LDAT_ACT=LV020Z0
FDAT_ACT=FPLAS90519LS1_2
BAS(#CP_PARAMS,0.3)
LIN XPLAS90519LS1_2
;ENDFOLD


;Movimimiento de busqueda con laser
;Search( , )

LIN_OFFS(XPLAS90519LS1_1, FPLAS90519LS1_1, 0, -200, 0, 0, 0, 0, #TOOL, 0.3, 50, 0.0)

;******************************;

;FOLD PTP pWB90519LS1 Vel=100 % PDAT_MESA Tool[10]:AMF1_G1000 Base[14]:BWB2S1;%{PE}%R 5.5.32,%MKUKATPBASIS,%CMOVE,%VPTP,%P 1:PTP, 2:pWB90519LS1, 3:, 5:100, 7:PDAT_MESA
$BWDSTART=FALSE
PDAT_ACT=PPDAT_MESA
FDAT_ACT=FpWB90519LS1
BAS(#PTP_PARAMS,100)
PTP XpWB90519LS1
;ENDFOLD

;*******************************************************
CASE 90521
;*******************************************************
;*** Utilizar para hacer touchup en ptp a continuacion ***;
; 1  Ejecutar Axis_Rob_Move
; 2  Hacer TouchUp en ptp
; 3  Eliminar Axis_Rob_Move y comentarios

Axis_Rob_Move(1.69,-82.8,66.93,14.32,12.14,193,70,50)

;FOLD PTP pWB90521LS1 Vel=100 % PDAT_MESA Tool[10]:AMF1_G1000 Base[14]:BWB2S1;%{PE}%R 5.5.32,%MKUKATPBASIS,%CMOVE,%VPTP,%P 1:PTP, 2:pWB90521LS1, 3:, 5:100, 7:PDAT_MESA
$BWDSTART=FALSE
PDAT_ACT=PPDAT_MESA
FDAT_ACT=FpWB90521LS1
BAS(#PTP_PARAMS,100)
PTP XpWB90521LS1
;ENDFOLD
;*********************************************************;

;***Axis_Rob_Move de ayuda para aproximarse a dejada ***;
; Borrar tras touchup en LIN de dejada
Axis_Rob_Move(-90.22,-57.13,49.23,-5.44,97.37,193.9,20,50)
;*******************************************************;

PTP_OFFS(XP90521LS1, FP90521LS1, 0, -450, 30, 0, 0, 0, #TOOL, 20, 50, 0.0)

Cicle_Grp_M1000 (Inic_Pla_Right)

;***borrar***;
cyltopos(prg_200)
halt
;************;

LIN_OFFS(XP90521LS1, FP90521LS1, 0, 0, 30, 0, 0, 0, #TOOL, 0.1, 50, 0.0)
LIN_OFFS(XP90521LS1, FP90521LS1, 0, 0, 15, 0, 0, 0, #TOOL, 0.1, 50, 0.0)

Cntr_Grp_M1000 (C05C06,RH)

;FOLD LIN P90521LS1 Vel=0.1 m/s LV020Z0 Tool[10]:AMF1_G1000 Base[14]:BWB2S1;%{PE}%R 5.5.32,%MKUKATPBASIS,%CMOVE,%VLIN,%P 1:LIN, 2:P90521LS1, 3:, 5:0.1, 7:V020Z0
$BWDSTART=FALSE
LDAT_ACT=LV020Z0
FDAT_ACT=FP90521LS1
BAS(#CP_PARAMS,0.1)
LIN XP90521LS1
;ENDFOLD

Cntr_Grp_M1000 (AMF09,RLS)
Cyltopos (PRG_51)
Cntr_Grp_M1000 (C07C08,RH)
Cyltopos (PRG_61)
Cntr_Grp_M1000 (AMF10,RLS)
Cntr_Grp_M1000 (C05C06,FREE)
Cntr_Grp_M1000 (C07C08,FREE)
Cyltopos(PRG_88)
LIN_REL{Z -20}#TOOL
Cyltopos (PRG_105)
LIN_REL{Z -30}#TOOL
Cyltopos (PRG_200)

;*** MOVIMIENTOS DE OFFSETS ***;

LIN_OFFS(XP90521LS1, FP90521LS1, 0, 0, -50, 0, 0, 0, #TOOL, 0.3, 50, 0.0)
LIN_OFFS(XP90521LS1, FP90521LS1, 0, -450, -50, 0, 0, 0, #TOOL, 0.3, 50, 0.0)


;******* MEDICION LASER *******;

LIN_OFFS(XPLAS90521LS1_1, FPLAS90521LS1_1, 0, -200, 0, 0, 0, 0, #TOOL, 0.3, 50, 0.0)

cyltopos (prg_61)

;FOLD LIN PLAS90521LS1_1 Vel=0.3 m/s LV020Z0 Tool[10]:AMF1_G1000 Base[14]:BWB2S1;%{PE}%R 5.5.32,%MKUKATPBASIS,%CMOVE,%VLIN,%P 1:LIN, 2:PLAS90521LS1_1, 3:, 5:0.3, 7:V020Z0
$BWDSTART=FALSE
LDAT_ACT=LV020Z0
FDAT_ACT=FPLAS90521LS1_1
BAS(#CP_PARAMS,0.3)
LIN XPLAS90521LS1_1
;ENDFOLD

;Movimimiento de busqueda con laser
;Search( , )

;FOLD LIN PLAS90521LS1_2 Vel=0.3 m/s LV020Z0 Tool[10]:AMF1_G1000 Base[14]:BWB2S1;%{PE}%R 5.5.32,%MKUKATPBASIS,%CMOVE,%VLIN,%P 1:LIN, 2:PLAS90521LS1_2, 3:, 5:0.3, 7:V020Z0
$BWDSTART=FALSE
LDAT_ACT=LV020Z0
FDAT_ACT=FPLAS90521LS1_2
BAS(#CP_PARAMS,0.3)
LIN XPLAS90521LS1_2
;ENDFOLD


;Movimimiento de busqueda con laser
;Search( , )

LIN_OFFS(XPLAS90521LS1_1, FPLAS90521LS1_1, 0, -200, 0, 0, 0, 0, #TOOL, 0.3, 50, 0.0)

;******************************;

;FOLD PTP pWB90521LS1 Vel=100 % PDAT_MESA Tool[10]:AMF1_G1000 Base[14]:BWB2S1;%{PE}%R 5.5.32,%MKUKATPBASIS,%CMOVE,%VPTP,%P 1:PTP, 2:pWB90521LS1, 3:, 5:100, 7:PDAT_MESA
$BWDSTART=FALSE
PDAT_ACT=PPDAT_MESA
FDAT_ACT=FpWB90521LS1
BAS(#PTP_PARAMS,100)
PTP XpWB90521LS1
;ENDFOLD

;*******************************************************
CASE 90523
;*******************************************************
;*** Utilizar para hacer touchup en ptp a continuacion ***;
; 1  Ejecutar Axis_Rob_Move
; 2  Hacer TouchUp en ptp
; 3  Eliminar Axis_Rob_Move y comentarios

Axis_Rob_Move(1.69,-82.8,66.93,14.32,12.14,193,70,50)

;FOLD PTP pWB90523LS1 Vel=100 % PDAT_MESA Tool[10]:AMF1_G1000 Base[14]:BWB2S1;%{PE}%R 5.5.32,%MKUKATPBASIS,%CMOVE,%VPTP,%P 1:PTP, 2:pWB90523LS1, 3:, 5:100, 7:PDAT_MESA
$BWDSTART=FALSE
PDAT_ACT=PPDAT_MESA
FDAT_ACT=FpWB90523LS1
BAS(#PTP_PARAMS,100)
PTP XpWB90523LS1
;ENDFOLD
;*********************************************************;

;***Axis_Rob_Move de ayuda para aproximarse a dejada ***;
; Borrar tras touchup en LIN de dejada
Axis_Rob_Move(-90.22,-57.13,49.23,-5.44,97.37,193.9,20,50)
;*******************************************************;

PTP_OFFS(XP90523LS1, FP90523LS1, 0, -450, 30, 0, 0, 0, #TOOL, 20, 50, 0.0)

Cicle_Grp_M1000 (Inic_Pla_Right)

;***borrar***;
cyltopos(prg_200)
halt
;************;

LIN_OFFS(XP90523LS1, FP90523LS1, 0, 0, 30, 0, 0, 0, #TOOL, 0.1, 50, 0.0)
LIN_OFFS(XP90523LS1, FP90523LS1, 0, 0, 15, 0, 0, 0, #TOOL, 0.1, 50, 0.0)

Cntr_Grp_M1000 (C05C06,RH)

;FOLD LIN P90523LS1 Vel=0.1 m/s LV020Z0 Tool[10]:AMF1_G1000 Base[14]:BWB2S1;%{PE}%R 5.5.32,%MKUKATPBASIS,%CMOVE,%VLIN,%P 1:LIN, 2:P90523LS1, 3:, 5:0.1, 7:V020Z0
$BWDSTART=FALSE
LDAT_ACT=LV020Z0
FDAT_ACT=FP90523LS1
BAS(#CP_PARAMS,0.1)
LIN XP90523LS1
;ENDFOLD

Cntr_Grp_M1000 (AMF09,RLS)
Cyltopos (PRG_51)
Cntr_Grp_M1000 (C07C08,RH)
Cyltopos (PRG_61)
Cntr_Grp_M1000 (AMF10,RLS)
Cntr_Grp_M1000 (C05C06,FREE)
Cntr_Grp_M1000 (C07C08,FREE)
Cyltopos(PRG_88)
LIN_REL{Z -20}#TOOL
Cyltopos (PRG_105)
LIN_REL{Z -30}#TOOL
Cyltopos (PRG_200)

;*** MOVIMIENTOS DE OFFSETS ***;

LIN_OFFS(XP90523LS1, FP90523LS1, 0, 0, -50, 0, 0, 0, #TOOL, 0.3, 50, 0.0)
LIN_OFFS(XP90523LS1, FP90523LS1, 0, -450, -50, 0, 0, 0, #TOOL, 0.3, 50, 0.0)


;******* MEDICION LASER *******;

LIN_OFFS(XPLAS90523LS1_1, FPLAS90523LS1_1, 0, -200, 0, 0, 0, 0, #TOOL, 0.3, 50, 0.0)

cyltopos (prg_61)

;FOLD LIN PLAS90523LS1_1 Vel=0.3 m/s LV020Z0 Tool[10]:AMF1_G1000 Base[14]:BWB2S1;%{PE}%R 5.5.32,%MKUKATPBASIS,%CMOVE,%VLIN,%P 1:LIN, 2:PLAS90523LS1_1, 3:, 5:0.3, 7:V020Z0
$BWDSTART=FALSE
LDAT_ACT=LV020Z0
FDAT_ACT=FPLAS90523LS1_1
BAS(#CP_PARAMS,0.3)
LIN XPLAS90523LS1_1
;ENDFOLD

;Movimimiento de busqueda con laser
;Search( , )

;FOLD LIN PLAS90523LS1_2 Vel=0.3 m/s LV020Z0 Tool[10]:AMF1_G1000 Base[14]:BWB2S1;%{PE}%R 5.5.32,%MKUKATPBASIS,%CMOVE,%VLIN,%P 1:LIN, 2:PLAS90523LS1_2, 3:, 5:0.3, 7:V020Z0
$BWDSTART=FALSE
LDAT_ACT=LV020Z0
FDAT_ACT=FPLAS90523LS1_2
BAS(#CP_PARAMS,0.3)
LIN XPLAS90523LS1_2
;ENDFOLD


;Movimimiento de busqueda con laser
;Search( , )

LIN_OFFS(XPLAS90523LS1_1, FPLAS90523LS1_1, 0, -200, 0, 0, 0, 0, #TOOL, 0.3, 50, 0.0)

;******************************;

;FOLD PTP pWB90523LS1 Vel=100 % PDAT_MESA Tool[10]:AMF1_G1000 Base[14]:BWB2S1;%{PE}%R 5.5.32,%MKUKATPBASIS,%CMOVE,%VPTP,%P 1:PTP, 2:pWB90523LS1, 3:, 5:100, 7:PDAT_MESA
$BWDSTART=FALSE
PDAT_ACT=PPDAT_MESA
FDAT_ACT=FpWB90523LS1
BAS(#PTP_PARAMS,100)
PTP XpWB90523LS1
;ENDFOLD

ENDSWITCH
END

--- nplacestr5LS1.dat ---
DEFDAT nplacestr5LS1
;FOLD EXTERNAL DECLARATIONS;%{PE}%MKUKATPBASIS,%CEXT,%VCOMMON,%P
;FOLD BASISTECH EXT;%{PE}%MKUKATPBASIS,%CEXT,%VEXT,%P
EXT  BAS (BAS_COMMAND  :IN,REAL  :IN )
DECL INT SUCCESS
;ENDFOLD (BASISTECH EXT)
;FOLD USER EXT;%{E}%MKUKATPUSER,%CEXT,%VEXT,%P
;Make here your modifications

;ENDFOLD (USER EXT)
;ENDFOLD (EXTERNAL DECLARATIONS)
DECL E6POS XpWB90501LS1={X 0,Y 0,Z 0,A 0,B 0,C 0,S 2,T 10,E1 0.0,E2 0.0,E3 0.0,E4 0.0,E5 0.0,E6 0.0}
DECL FDAT FpWB90501LS1={TOOL_NO 10,BASE_NO 14,IPO_FRAME #BASE,POINT2[] " ",TQ_STATE FALSE}
;
DECL E6POS XP90501LS1={X 0,Y 0,Z 0,A 0,B 0,C 0,S 2,T 10,E1 0.0,E2 0.0,E3 0.0,E4 0.0,E5 0.0,E6 0.0}
DECL FDAT FP90501LS1={TOOL_NO 10,BASE_NO 14,IPO_FRAME #BASE,POINT2[] " ",TQ_STATE FALSE}
;
DECL E6POS XPLAS90501LS1_1={X 0,Y 0,Z 0,A 0,B 0,C 0,S 2,T 10,E1 0.0,E2 0.0,E3 0.0,E4 0.0,E5 0.0,E6 0.0}
DECL FDAT FPLAS90501LS1_1={TOOL_NO 10,BASE_NO 14,IPO_FRAME #BASE,POINT2[] " ",TQ_STATE FALSE}
DECL E6POS XPLAS90501LS1_2={X 0,Y 0,Z 0,A 0,B 0,C 0,S 2,T 10,E1 0.0,E2 0.0,E3 0.0,E4 0.0,E5 0.0,E6 0.0}
DECL FDAT FPLAS90501LS1_2={TOOL_NO 10,BASE_NO 14,IPO_FRAME #BASE,POINT2[] " ",TQ_STATE FALSE}
;
DECL E6POS XpWB90503LS1={X 0,Y 0,Z 0,A 0,B 0,C 0,S 2,T 10,E1 0.0,E2 0.0,E3 0.0,E4 0.0,E5 0.0,E6 0.0}
DECL FDAT FpWB90503LS1={TOOL_NO 10,BASE_NO 14,IPO_FRAME #BASE,POINT2[] " ",TQ_STATE FALSE}
;
DECL E6POS XP90503LS1={X 0,Y 0,Z 0,A 0,B 0,C 0,S 2,T 10,E1 0.0,E2 0.0,E3 0.0,E4 0.0,E5 0.0,E6 0.0}
DECL FDAT FP90503LS1={TOOL_NO 10,BASE_NO 14,IPO_FRAME #BASE,POINT2[] " ",TQ_STATE FALSE}
;
DECL E6POS XPLAS90503LS1_1={X 0,Y 0,Z 0,A 0,B 0,C 0,S 2,T 10,E1 0.0,E2 0.0,E3 0.0,E4 0.0,E5 0.0,E6 0.0}
DECL FDAT FPLAS90503LS1_1={TOOL_NO 10,BASE_NO 14,IPO_FRAME #BASE,POINT2[] " ",TQ_STATE FALSE}
DECL E6POS XPLAS90503LS1_2={X 0,Y 0,Z 0,A 0,B 0,C 0,S 2,T 10,E1 0.0,E2 0.0,E3 0.0,E4 0.0,E5 0.0,E6 0.0}
DECL FDAT FPLAS90503LS1_2={TOOL_NO 10,BASE_NO 14,IPO_FRAME #BASE,POINT2[] " ",TQ_STATE FALSE}
;
DECL E6POS XpWB90505LS1={X 0,Y 0,Z 0,A 0,B 0,C 0,S 2,T 10,E1 0.0,E2 0.0,E3 0.0,E4 0.0,E5 0.0,E6 0.0}
DECL FDAT FpWB90505LS1={TOOL_NO 10,BASE_NO 14,IPO_FRAME #BASE,POINT2[] " ",TQ_STATE FALSE}
;
DECL E6POS XP90505LS1={X 0,Y 0,Z 0,A 0,B 0,C 0,S 2,T 10,E1 0.0,E2 0.0,E3 0.0,E4 0.0,E5 0.0,E6 0.0}
DECL FDAT FP90505LS1={TOOL_NO 10,BASE_NO 14,IPO_FRAME #BASE,POINT2[] " ",TQ_STATE FALSE}
;
DECL E6POS XPLAS90505LS1_1={X 0,Y 0,Z 0,A 0,B 0,C 0,S 2,T 10,E1 0.0,E2 0.0,E3 0.0,E4 0.0,E5 0.0,E6 0.0}
DECL FDAT FPLAS90505LS1_1={TOOL_NO 10,BASE_NO 14,IPO_FRAME #BASE,POINT2[] " ",TQ_STATE FALSE}
DECL E6POS XPLAS90505LS1_2={X 0,Y 0,Z 0,A 0,B 0,C 0,S 2,T 10,E1 0.0,E2 0.0,E3 0.0,E4 0.0,E5 0.0,E6 0.0}
DECL FDAT FPLAS90505LS1_2={TOOL_NO 10,BASE_NO 14,IPO_FRAME #BASE,POINT2[] " ",TQ_STATE FALSE}
;
DECL E6POS XpWB90507LS1={X 0,Y 0,Z 0,A 0,B 0,C 0,S 2,T 10,E1 0.0,E2 0.0,E3 0.0,E4 0.0,E5 0.0,E6 0.0}
DECL FDAT FpWB90507LS1={TOOL_NO 10,BASE_NO 14,IPO_FRAME #BASE,POINT2[] " ",TQ_STATE FALSE}
;
DECL E6POS XP90507LS1={X 0,Y 0,Z 0,A 0,B 0,C 0,S 2,T 10,E1 0.0,E2 0.0,E3 0.0,E4 0.0,E5 0.0,E6 0.0}
DECL FDAT FP90507LS1={TOOL_NO 10,BASE_NO 14,IPO_FRAME #BASE,POINT2[] " ",TQ_STATE FALSE}
;
DECL E6POS XPLAS90507LS1_1={X 0,Y 0,Z 0,A 0,B 0,C 0,S 2,T 10,E1 0.0,E2 0.0,E3 0.0,E4 0.0,E5 0.0,E6 0.0}
DECL FDAT FPLAS90507LS1_1={TOOL_NO 10,BASE_NO 14,IPO_FRAME #BASE,POINT2[] " ",TQ_STATE FALSE}
DECL E6POS XPLAS90507LS1_2={X 0,Y 0,Z 0,A 0,B 0,C 0,S 2,T 10,E1 0.0,E2 0.0,E3 0.0,E4 0.0,E5 0.0,E6 0.0}
DECL FDAT FPLAS90507LS1_2={TOOL_NO 10,BASE_NO 14,IPO_FRAME #BASE,POINT2[] " ",TQ_STATE FALSE}
;
DECL E6POS XpWB90509LS1={X 0,Y 0,Z 0,A 0,B 0,C 0,S 2,T 10,E1 0.0,E2 0.0,E3 0.0,E4 0.0,E5 0.0,E6 0.0}
DECL FDAT FpWB90509LS1={TOOL_NO 10,BASE_NO 14,IPO_FRAME #BASE,POINT2[] " ",TQ_STATE FALSE}
;
DECL E6POS XP90509LS1={X 0,Y 0,Z 0,A 0,B 0,C 0,S 2,T 10,E1 0.0,E2 0.0,E3 0.0,E4 0.0,E5 0.0,E6 0.0}
DECL FDAT FP90509LS1={TOOL_NO 10,BASE_NO 14,IPO_FRAME #BASE,POINT2[] " ",TQ_STATE FALSE}
;
DECL E6POS XPLAS90509LS1_1={X 0,Y 0,Z 0,A 0,B 0,C 0,S 2,T 10,E1 0.0,E2 0.0,E3 0.0,E4 0.0,E5 0.0,E6 0.0}
DECL FDAT FPLAS90509LS1_1={TOOL_NO 10,BASE_NO 14,IPO_FRAME #BASE,POINT2[] " ",TQ_STATE FALSE}
DECL E6POS XPLAS90509LS1_2={X 0,Y 0,Z 0,A 0,B 0,C 0,S 2,T 10,E1 0.0,E2 0.0,E3 0.0,E4 0.0,E5 0.0,E6 0.0}
DECL FDAT FPLAS90509LS1_2={TOOL_NO 10,BASE_NO 14,IPO_FRAME #BASE,POINT2[] " ",TQ_STATE FALSE}
;
DECL E6POS XpWB90511LS1={X 0,Y 0,Z 0,A 0,B 0,C 0,S 2,T 10,E1 0.0,E2 0.0,E3 0.0,E4 0.0,E5 0.0,E6 0.0}
DECL FDAT FpWB90511LS1={TOOL_NO 10,BASE_NO 14,IPO_FRAME #BASE,POINT2[] " ",TQ_STATE FALSE}
;
DECL E6POS XP90511LS1={X 0,Y 0,Z 0,A 0,B 0,C 0,S 2,T 10,E1 0.0,E2 0.0,E3 0.0,E4 0.0,E5 0.0,E6 0.0}
DECL FDAT FP90511LS1={TOOL_NO 10,BASE_NO 14,IPO_FRAME #BASE,POINT2[] " ",TQ_STATE FALSE}
;
DECL E6POS XPLAS90511LS1_1={X 0,Y 0,Z 0,A 0,B 0,C 0,S 2,T 10,E1 0.0,E2 0.0,E3 0.0,E4 0.0,E5 0.0,E6 0.0}
DECL FDAT FPLAS90511LS1_1={TOOL_NO 10,BASE_NO 14,IPO_FRAME #BASE,POINT2[] " ",TQ_STATE FALSE}
DECL E6POS XPLAS90511LS1_2={X 0,Y 0,Z 0,A 0,B 0,C 0,S 2,T 10,E1 0.0,E2 0.0,E3 0.0,E4 0.0,E5 0.0,E6 0.0}
DECL FDAT FPLAS90511LS1_2={TOOL_NO 10,BASE_NO 14,IPO_FRAME #BASE,POINT2[] " ",TQ_STATE FALSE}
;
DECL E6POS XpWB90513LS1={X 0,Y 0,Z 0,A 0,B 0,C 0,S 2,T 10,E1 0.0,E2 0.0,E3 0.0,E4 0.0,E5 0.0,E6 0.0}
DECL FDAT FpWB90513LS1={TOOL_NO 10,BASE_NO 14,IPO_FRAME #BASE,POINT2[] " ",TQ_STATE FALSE}
;
DECL E6POS XP90513LS1={X 0,Y 0,Z 0,A 0,B 0,C 0,S 2,T 10,E1 0.0,E2 0.0,E3 0.0,E4 0.0,E5 0.0,E6 0.0}
DECL FDAT FP90513LS1={TOOL_NO 10,BASE_NO 14,IPO_FRAME #BASE,POINT2[] " ",TQ_STATE FALSE}
;
DECL E6POS XPLAS90513LS1_1={X 0,Y 0,Z 0,A 0,B 0,C 0,S 2,T 10,E1 0.0,E2 0.0,E3 0.0,E4 0.0,E5 0.0,E6 0.0}
DECL FDAT FPLAS90513LS1_1={TOOL_NO 10,BASE_NO 14,IPO_FRAME #BASE,POINT2[] " ",TQ_STATE FALSE}
DECL E6POS XPLAS90513LS1_2={X 0,Y 0,Z 0,A 0,B 0,C 0,S 2,T 10,E1 0.0,E2 0.0,E3 0.0,E4 0.0,E5 0.0,E6 0.0}
DECL FDAT FPLAS90513LS1_2={TOOL_NO 10,BASE_NO 14,IPO_FRAME #BASE,POINT2[] " ",TQ_STATE FALSE}
;
DECL E6POS XpWB90515LS1={X 0,Y 0,Z 0,A 0,B 0,C 0,S 2,T 10,E1 0.0,E2 0.0,E3 0.0,E4 0.0,E5 0.0,E6 0.0}
DECL FDAT FpWB90515LS1={TOOL_NO 10,BASE_NO 14,IPO_FRAME #BASE,POINT2[] " ",TQ_STATE FALSE}
;
DECL E6POS XP90515LS1={X 0,Y 0,Z 0,A 0,B 0,C 0,S 2,T 10,E1 0.0,E2 0.0,E3 0.0,E4 0.0,E5 0.0,E6 0.0}
DECL FDAT FP90515LS1={TOOL_NO 10,BASE_NO 14,IPO_FRAME #BASE,POINT2[] " ",TQ_STATE FALSE}
;
DECL E6POS XPLAS90515LS1_1={X 0,Y 0,Z 0,A 0,B 0,C 0,S 2,T 10,E1 0.0,E2 0.0,E3 0.0,E4 0.0,E5 0.0,E6 0.0}
DECL FDAT FPLAS90515LS1_1={TOOL_NO 10,BASE_NO 14,IPO_FRAME #BASE,POINT2[] " ",TQ_STATE FALSE}
DECL E6POS XPLAS90515LS1_2={X 0,Y 0,Z 0,A 0,B 0,C 0,S 2,T 10,E1 0.0,E2 0.0,E3 0.0,E4 0.0,E5 0.0,E6 0.0}
DECL FDAT FPLAS90515LS1_2={TOOL_NO 10,BASE_NO 14,IPO_FRAME #BASE,POINT2[] " ",TQ_STATE FALSE}
;
DECL E6POS XpWB90517LS1={X 0,Y 0,Z 0,A 0,B 0,C 0,S 2,T 10,E1 0.0,E2 0.0,E3 0.0,E4 0.0,E5 0.0,E6 0.0}
DECL FDAT FpWB90517LS1={TOOL_NO 10,BASE_NO 14,IPO_FRAME #BASE,POINT2[] " ",TQ_STATE FALSE}
;
DECL E6POS XP90517LS1={X 0,Y 0,Z 0,A 0,B 0,C 0,S 2,T 10,E1 0.0,E2 0.0,E3 0.0,E4 0.0,E5 0.0,E6 0.0}
DECL FDAT FP90517LS1={TOOL_NO 10,BASE_NO 14,IPO_FRAME #BASE,POINT2[] " ",TQ_STATE FALSE}
;
DECL E6POS XPLAS90517LS1_1={X 0,Y 0,Z 0,A 0,B 0,C 0,S 2,T 10,E1 0.0,E2 0.0,E3 0.0,E4 0.0,E5 0.0,E6 0.0}
DECL FDAT FPLAS90517LS1_1={TOOL_NO 10,BASE_NO 14,IPO_FRAME #BASE,POINT2[] " ",TQ_STATE FALSE}
DECL E6POS XPLAS90517LS1_2={X 0,Y 0,Z 0,A 0,B 0,C 0,S 2,T 10,E1 0.0,E2 0.0,E3 0.0,E4 0.0,E5 0.0,E6 0.0}
DECL FDAT FPLAS90517LS1_2={TOOL_NO 10,BASE_NO 14,IPO_FRAME #BASE,POINT2[] " ",TQ_STATE FALSE}
;
DECL E6POS XpWB90519LS1={X 0,Y 0,Z 0,A 0,B 0,C 0,S 2,T 10,E1 0.0,E2 0.0,E3 0.0,E4 0.0,E5 0.0,E6 0.0}
DECL FDAT FpWB90519LS1={TOOL_NO 10,BASE_NO 14,IPO_FRAME #BASE,POINT2[] " ",TQ_STATE FALSE}
;
DECL E6POS XP90519LS1={X 0,Y 0,Z 0,A 0,B 0,C 0,S 2,T 10,E1 0.0,E2 0.0,E3 0.0,E4 0.0,E5 0.0,E6 0.0}
DECL FDAT FP90519LS1={TOOL_NO 10,BASE_NO 14,IPO_FRAME #BASE,POINT2[] " ",TQ_STATE FALSE}
;
DECL E6POS XPLAS90519LS1_1={X 0,Y 0,Z 0,A 0,B 0,C 0,S 2,T 10,E1 0.0,E2 0.0,E3 0.0,E4 0.0,E5 0.0,E6 0.0}
DECL FDAT FPLAS90519LS1_1={TOOL_NO 10,BASE_NO 14,IPO_FRAME #BASE,POINT2[] " ",TQ_STATE FALSE}
DECL E6POS XPLAS90519LS1_2={X 0,Y 0,Z 0,A 0,B 0,C 0,S 2,T 10,E1 0.0,E2 0.0,E3 0.0,E4 0.0,E5 0.0,E6 0.0}
DECL FDAT FPLAS90519LS1_2={TOOL_NO 10,BASE_NO 14,IPO_FRAME #BASE,POINT2[] " ",TQ_STATE FALSE}
;
DECL E6POS XpWB90521LS1={X 0,Y 0,Z 0,A 0,B 0,C 0,S 2,T 10,E1 0.0,E2 0.0,E3 0.0,E4 0.0,E5 0.0,E6 0.0}
DECL FDAT FpWB90521LS1={TOOL_NO 10,BASE_NO 14,IPO_FRAME #BASE,POINT2[] " ",TQ_STATE FALSE}
;
DECL E6POS XP90521LS1={X 0,Y 0,Z 0,A 0,B 0,C 0,S 2,T 10,E1 0.0,E2 0.0,E3 0.0,E4 0.0,E5 0.0,E6 0.0}
DECL FDAT FP90521LS1={TOOL_NO 10,BASE_NO 14,IPO_FRAME #BASE,POINT2[] " ",TQ_STATE FALSE}
;
DECL E6POS XPLAS90521LS1_1={X 0,Y 0,Z 0,A 0,B 0,C 0,S 2,T 10,E1 0.0,E2 0.0,E3 0.0,E4 0.0,E5 0.0,E6 0.0}
DECL FDAT FPLAS90521LS1_1={TOOL_NO 10,BASE_NO 14,IPO_FRAME #BASE,POINT2[] " ",TQ_STATE FALSE}
DECL E6POS XPLAS90521LS1_2={X 0,Y 0,Z 0,A 0,B 0,C 0,S 2,T 10,E1 0.0,E2 0.0,E3 0.0,E4 0.0,E5 0.0,E6 0.0}
DECL FDAT FPLAS90521LS1_2={TOOL_NO 10,BASE_NO 14,IPO_FRAME #BASE,POINT2[] " ",TQ_STATE FALSE}
;
DECL E6POS XpWB90523LS1={X 0,Y 0,Z 0,A 0,B 0,C 0,S 2,T 10,E1 0.0,E2 0.0,E3 0.0,E4 0.0,E5 0.0,E6 0.0}
DECL FDAT FpWB90523LS1={TOOL_NO 10,BASE_NO 14,IPO_FRAME #BASE,POINT2[] " ",TQ_STATE FALSE}
;
DECL E6POS XP90523LS1={X 0,Y 0,Z 0,A 0,B 0,C 0,S 2,T 10,E1 0.0,E2 0.0,E3 0.0,E4 0.0,E5 0.0,E6 0.0}
DECL FDAT FP90523LS1={TOOL_NO 10,BASE_NO 14,IPO_FRAME #BASE,POINT2[] " ",TQ_STATE FALSE}
;
DECL E6POS XPLAS90523LS1_1={X 0,Y 0,Z 0,A 0,B 0,C 0,S 2,T 10,E1 0.0,E2 0.0,E3 0.0,E4 0.0,E5 0.0,E6 0.0}
DECL FDAT FPLAS90523LS1_1={TOOL_NO 10,BASE_NO 14,IPO_FRAME #BASE,POINT2[] " ",TQ_STATE FALSE}
DECL E6POS XPLAS90523LS1_2={X 0,Y 0,Z 0,A 0,B 0,C 0,S 2,T 10,E1 0.0,E2 0.0,E3 0.0,E4 0.0,E5 0.0,E6 0.0}
DECL FDAT FPLAS90523LS1_2={TOOL_NO 10,BASE_NO 14,IPO_FRAME #BASE,POINT2[] " ",TQ_STATE FALSE}
;
ENDDAT
